Yaskawa INFORM job: FRONT_SEARCH_-90ST-2_5140.JBI

/JOB
//NAME FRONT_SEARCH_-90ST-2_5140
///FOLDERNAME 02-SKRZYNIE_JOBS
//POS
///NPOS 49,49,0,7,0,0
///TOOL 0
///POSTYPE PULSE
///PULSE
C00000=-14334,-10708,45002,-95286,-40321,-4878
C00001=-1,-11355,44471,-89821,-32839,-4429
C00002=51470,-3981,47579,-58794,-5299,-8788
C00003=55570,1468,42458,-7386,-9208,-33373
C00004=67803,1091,42035,59104,-16935,-61314
C00005=66620,9721,53664,53490,-17138,-58745
C00006=65132,11491,55975,50657,-16585,-57605
C00007=66620,9721,53664,53490,-17138,-58745
C00008=67271,11853,56546,53440,-17675,-58611
C00009=54816,3282,46487,30906,-12207,-49746
C00010=54816,6101,53312,25756,-14460,-47262
C00011=57034,1893,43594,38914,-12219,-53230
C00012=38808,-5107,37135,-20098,-11081,-27963
C00013=36418,-5540,36288,-27687,-11438,-24719
C00014=35573,-4115,37713,-30259,-11607,-23622
C00015=37318,-4451,38463,-23712,-11808,-26477
C00016=36649,-2628,43243,-22183,-13723,-27325
C00017=36418,-5540,36288,-27687,-11438,-24719
C00018=12465,-20824,6291,-123875,-11964,11912
C00019=12465,-20824,6291,-123875,-11964,11912
C00020=12194,-19644,7182,-124437,-12272,12151
C00021=13120,-20758,6341,-124984,-11645,12518
C00022=12783,-19506,9715,-119026,-11009,9627
C00023=12465,-20824,6291,-123875,-11964,11912
C00024=-19334,-23740,-4461,-126950,-27208,2994
C00025=-19334,-23740,-4461,-126950,-27208,2994
C00026=-18876,-22402,-3481,-127715,-27199,3442
C00027=-19334,-23740,-4461,-126950,-27208,2994
C00028=-19334,-22649,-1366,-125024,-26367,1978
C00029=-19334,-23740,-4461,-126950,-27208,2994
C00030=-19623,-34877,-16768,-124729,-29078,-51940
C00031=-23953,-24934,-2154,-142846,-12846,-40273
C00032=-24662,-23944,-606,-140607,-12835,-41421
C00033=-24166,-22898,142,-142287,-12883,-40561
C00034=-24266,-23113,-13,-141949,-12872,-40733
C00035=-24266,-22239,2374,-139471,-12061,-41925
C00036=-24665,-23955,-613,-140592,-12836,-41426
C00037=-57975,-11422,9680,-117300,-24442,-51599
C00038=-57975,-11422,9680,-117300,-24442,-51599
C00039=-56559,-9965,11026,-118413,-23739,-50892
C00040=-57975,-11422,9680,-117300,-24442,-51599
C00041=-57975,-9264,15839,-112245,-23199,-54199
C00042=-51982,-12153,15004,-104816,-14508,-60674
C00043=-56524,-9302,17607,-103995,-17398,-61581
C00044=-55122,-10973,14720,-110381,-19153,-56434
C00045=-46873,-31323,-15655,-127144,-23194,-47707
C00046=-53252,-41973,-2905,-102185,-37459,-42403
C00047=0,-35574,42087,-36666,-9339,-1809
C00048=0,-52278,40443,0,6873,-1
BC00000=806966
BC00001=874451
BC00002=918461
BC00003=970051
BC00004=970051
BC00005=970051
BC00006=970051
BC00007=970051
BC00008=970051
BC00009=970052
BC00010=970052
BC00011=970052
BC00012=970052
BC00013=970052
BC00014=970052
BC00015=970052
BC00016=970052
BC00017=970052
BC00018=970052
BC00019=970052
BC00020=970052
BC00021=970052
BC00022=970052
BC00023=970052
BC00024=970052
BC00025=970052
BC00026=970052
BC00027=970052
BC00028=970052
BC00029=970052
BC00030=970052
BC00031=970052
BC00032=970052
BC00033=970052
BC00034=970052
BC00035=970052
BC00036=970052
BC00037=970049
BC00038=970049
BC00039=970049
BC00040=970049
BC00041=970049
BC00042=970049
BC00043=970049
BC00044=970050
BC00045=970050
BC00046=911348
BC00047=796997
BC00048=790120
///POSTYPE BASE
///RECTAN
///RCONF 1,0,0,0,0,0,0,0,0,0,0,0,0,0,0,0,0,0,0,0,0,0,0,0
P00006=0.000,0.000,0.000,0.0000,0.0000,0.0000
P00500=2.332,-5.281,-1.258,0.0000,0.0000,0.0000
///RCONF 0,0,0,0,0,0,0,0,0,0,0,0,0,0,0,0,0,0,0,0,0,0,0,0
P00501=-2.026,0.009,3.534,0.0000,0.0000,0.0000
///RCONF 1,0,0,0,0,0,0,0,0,0,0,0,0,0,0,0,0,0,0,0,0,0,0,0
P00502=-2.023,0.001,1.732,0.0000,0.0000,0.0000
P00503=0.138,-0.044,1.539,0.0000,0.0000,0.0000
P00504=-0.309,-0.010,1.636,0.0000,0.0000,0.0000
P00505=0.999,-9.916,8.214,0.0000,0.0000,0.0000
//INST
///DATE 2024/06/04 21:27
///ATTR SC,RW
///GROUP1 RB1,BS1
NOP
MOVJ C00000 BC00000 VJ=50.00
MOVJ C00001 BC00001 VJ=70.00
MOVJ C00002 BC00002 VJ=60.00
MOVJ C00003 BC00003 VJ=50.00
'::::::::::::::::::::::::::::::::
'W21 P
'::::::::::::::::::::::::::::::::
MOVL C00004 BC00004 V=333.3
MOVL C00005 BC00005 V=166.7 PL=0
REFP 3 C00006 BC00006
CALL JOB:SEARCH-R1
SET P0500 P0006
SFTON P0500
MOVL C00007 BC00007 V=166.7 PL=0
REFP 3 C00008 BC00008
CALL JOB:SEARCH-R1
SET P0500 P0006
SFTON P0500
MOVL C00009 BC00009 V=166.7 PL=0
REFP 3 C00010 BC00010
CALL JOB:SEARCH-R1
SET P0500 P0006
SFTOF
MOVL C00011 BC00011 V=166.7
'::::::::::::::::::::::::::::::::
'W21 L
'::::::::::::::::::::::::::::::::
MOVL C00012 BC00012 V=500.0
MOVL C00013 BC00013 V=166.7 PL=0
REFP 3 C00014 BC00014
CALL JOB:SEARCH-R1
SET P0501 P0006
SFTON P0501
MOVL C00015 BC00015 V=166.7 PL=0
REFP 3 C00016 BC00016
CALL JOB:SEARCH-R1
SET P0501 P0006
SFTON P0501
MOVL C00017 BC00017 V=166.7 PL=0
SFTOF
'::::::::::::::::::::::::::::::::
'W20 P
'::::::::::::::::::::::::::::::::
MOVL C00018 BC00018 V=500.0
MOVL C00019 BC00019 V=166.7 PL=0
REFP 3 C00020 BC00020
CALL JOB:SEARCH-R1
SET P0502 P0006
SFTON P0502
MOVL C00021 BC00021 V=166.7 PL=0
REFP 3 C00022 BC00022
CALL JOB:SEARCH-R1
SET P0502 P0006
SFTON P0502
MOVL C00023 BC00023 V=166.7 PL=0
SFTOF
'::::::::::::::::::::::::::::::::
'W20 L
'::::::::::::::::::::::::::::::::
MOVL C00024 BC00024 V=416.7
MOVL C00025 BC00025 V=166.7 PL=0
REFP 3 C00026 BC00026
CALL JOB:SEARCH-R1
SET P0503 P0006
SFTON P0503
MOVL C00027 BC00027 V=133.3 PL=0
REFP 3 C00028 BC00028
CALL JOB:SEARCH-R1
SET P0503 P0006
SFTON P0503
MOVL C00029 BC00029 V=166.7 PL=0
SFTOF
'::::::::::::::::::::::::::::::::
'W22 P
'::::::::::::::::::::::::::::::::
MOVL C00030 BC00030 V=166.7
MOVL C00031 BC00031 V=500.0
MOVL C00032 BC00032 V=166.7 PL=0
REFP 3 C00033 BC00033
CALL JOB:SEARCH-R1
SET P0504 P0006
SFTON P0504
MOVL C00034 BC00034 V=166.7 PL=0
REFP 3 C00035 BC00035
CALL JOB:SEARCH-R1
SET P0504 P0006
SFTON P0504
MOVL C00036 BC00036 V=166.7 PL=0
SFTOF
'::::::::::::::::::::::::::::::::
'W22 L
'::::::::::::::::::::::::::::::::
MOVL C00037 BC00037 V=416.7
MOVL C00038 BC00038 V=166.7 PL=0
REFP 3 C00039 BC00039
CALL JOB:SEARCH-R1
SET P0505 P0006
SFTON P0505
MOVL C00040 BC00040 V=166.7 PL=0
REFP 3 C00041 BC00041
CALL JOB:SEARCH-R1
SET P0505 P0006
SFTON P0505
MOVL C00042 BC00042 V=166.7 PL=0
REFP 3 C00043 BC00043
CALL JOB:SEARCH-R1
SET P0505 P0006
SFTOF
MOVL C00044 BC00044 V=83.3
MOVL C00045 BC00045 V=500.0
MOVJ C00046 BC00046 VJ=50.00
MOVJ C00047 BC00047 VJ=80.00
MOVJ C00048 BC00048 VJ=80.00
END
